(* IEC 61131-3 sources: CannyIEC/extracted_st/library_information/getlibversion, 1 file *)

(* ---- GetLibVersion.st ---- *)
(* --- Interface --- *)
// This function has been automatically generated from the project information.
FUNCTION GetLibVersion : VERSION
VAR_INPUT

END_VAR
(* --- Implementation --- *)
GetLibVersion.uiMajor := 0;
GetLibVersion.uiMinor := 1;
GetLibVersion.uiServicePack := 11;
GetLibVersion.uiPatch := 10;
